VAR_GLOBAL
//STOP			: 	BOOL;		//安全模块输出停


//mStart	: 	BOOL;


//mStop		:	BOOL;


//ZPulseSignalX	AT%I* 	:BOOL;


//ZPulseSignalY	AT%I* 	:BOOL;


//ZPulseSignalZ	AT%I* 	:BOOL;


//	bLimitHomeX:	BOOL;


//	bLimitHomeY:	BOOL;


//	bLimitHomeZ:	BOOL;


//	bPulseHomeX:	BOOL;


//	bPulseHomeY:	BOOL;


//	bPulseHomeZ:	BOOL;


//	bFinishHomeX:	BOOL;


//	bFinishHomeY:	BOOL;


//	bFinishHomeZ:	BOOL;


    AxisN               : AXIS_REF;
    CamInOutX           : ,;
    CamOutOutX, CamInOutY , CamOutOutY ST_McOutputs;
    safetySignal        : BOOL;
    SysStep             : INT; //系统状态步


aStep             : INT; //自动状态步



rAdvancedDonePos : LREAL;
    bCamInX             : BOOL;
    bCamInY             : BOOL;
    bCamOutX            : BOOL;
    bCamOutY            : BOOL;
    bReadyX             : BOOL;
    bReadyY             : BOOL;
    ton1                : ton;
    sig                 : BOOL;
END_VAR

(* stored: Version 1.1.0.1, ProductVersion 3.1.4024.12
   GVL GVL_Variables: Id {766d8d5b-91a3-46a8-ab61-270224db8376} *)
